(* IEC 61131-3 sources: RL_MAR/experiments/comparison/llm4plc/results/gpt-4o_20260507_114630/20260507_120937, 1 file *)

(* ---- generated_code_iteration_0.st ---- *)
plaintext
START_ST
FUNCTION_BLOCK FB_ThresholdAccumulator
VAR_INPUT
    i : INT; // Input value to be processed
END_VAR

VAR_OUTPUT
    o : INT; // Output value based on the logic
END_VAR

VAR
    s1 : INT; // Intermediate variable for calculations
END_VAR

// Initialize s1 to 0 at the start of the function block execution
s1 := 0;

// Check if the input i is greater than 0
IF i > 0 THEN
    s1 := s1 + i; // Add the value of i to s1
END_IF;

// Check if s1 equals 42 after the first condition
IF s1 = 42 THEN
    s1 := s1 + 8000; // Add 8000 to s1
END_IF;

// Determine the output o based on the value of s1
IF s1 < 0 THEN
    o := 0; // Set output to 0 if s1 is less than 0
ELSE
    o := s1; // Set output to the current value of s1 otherwise
END_IF;

END_FUNCTION_BLOCK
END_ST
